KUKA KRL data list: e_fraes_1.dat

&ACCESS RVP2
&REL 8
&COMMENT Fresa C1
&PARAM DISKPATH = KRC:\R1\Program
&PARAM TEMPLATE = C:\KRC\Roboter\Template\vorgabe
&PARAM EDITMASK = *
DEFDAT  e_fraes_1
;FOLD EXTERNAL DECLARATIONS;%{PE}%MKUKATPBASIS,%CEXT,%VCOMMON,%P
;FOLD GRIPPERTECH EXT
EXT  H50 (INT  :IN,INT  :IN,INT  :IN,GRP_TYP  :IN )
;ENDFOLD (GRIPPERTECH EXT)
;FOLD SPOTTECH EXT
EXT  USERSPOT (S_COMMAND  :IN,SPOT_TYPE  :IN )
;ENDFOLD (SPOTTECH EXT)
;FOLD BASISTECH EXT;%{PE}%MKUKATPBASIS,%CEXT,%VEXT,%P
EXT  BAS (BAS_COMMAND  :IN,REAL  :IN )
DECL INT SUCCESS
;ENDFOLD (BASISTECH EXT)
;FOLD USER EXT;%{E}%MKUKATPUSER,%CEXT,%VEXT,%P
;Make your modifications here

;ENDFOLD (USER EXT)
;ENDFOLD (EXTERNAL DECLARATIONS)

DECL E6POS XLHP010={X 388.052307,Y 1486.41003,Z 838.34668,A 150.907806,B -0.182968304,C -18.4479904,S 2,T 3,E1 0.0,E2 0.0,E3 0.0,E4 0.0,E5 0.0,E6 0.0}
DECL FDAT FLHP010={TOOL_NO 1,BASE_NO 0,IPO_FRAME #BASE}
DECL PDAT PPDAT1={VEL 100.0,ACC 100.0,APO_DIST 20.0,APO_MODE #CDIS}
DECL E6POS XLHP015={X 384.866791,Y 1472.83899,Z 444.33551,A -149.197906,B 0.240399107,C -3.14899206,S 18,T 11,E1 0.0,E2 0.0,E3 0.0,E4 0.0,E5 0.0,E6 0.0}
DECL FDAT FLHP015={TOOL_NO 1,BASE_NO 0,IPO_FRAME #BASE}
DECL PDAT PPDAT2={VEL 100.0,ACC 100.0,APO_DIST 10.0}
DECL E6POS XLHP020={X 309.223694,Y 1602.80103,Z 250.550003,A -134.665497,B -0.498555809,C -1.271559,S 18,T 11,E1 0.0,E2 0.0,E3 0.0,E4 0.0,E5 0.0,E6 0.0}
DECL FDAT FLHP020={TOOL_NO 1,BASE_NO 0,IPO_FRAME #BASE}
DECL PDAT PPDAT3={VEL 100.0,ACC 100.0,APO_DIST 5.0,APO_MODE #CDIS}
DECL E6POS XLHP025={X 98.0119705,Y 1699.85095,Z 256.256805,A -134.662704,B -0.490130603,C -1.27114701,S 18,T 11,E1 0.0,E2 0.0,E3 0.0,E4 0.0,E5 0.0,E6 0.0}
DECL FDAT FLHP025={TOOL_NO 1,BASE_NO 0,IPO_FRAME #BASE}
DECL LDAT LCPDAT1={VEL 2.0,ACC 100.0,APO_DIST 2.0,APO_FAC 50.0}
DECL FDAT FDress1={TOOL_NO 1,BASE_NO 0,IPO_FRAME #BASE}
DECL E6POS XDress1={X 99.6608887,Y 1696.71301,Z 300.036499,A -134.662994,B -0.49089241,C -1.27011204,S 18,T 11,E1 0.0,E2 0.0,E3 0.0,E4 0.0,E5 0.0,E6 0.0}
DECL E6POS XPFRESA={X 102.833801,Y 1696.37195,Z 300.660889,A -134.662903,B -0.489995897,C -1.26936698,S 18,T 11,E1 0.0,E2 0.0,E3 0.0,E4 0.0,E5 0.0,E6 0.0}
DECL FDAT Fpfresa={TOOL_NO 1,BASE_NO 0,IPO_FRAME #BASE}
DECL LDAT LCPDAT2={VEL 2.0,ACC 100.0,APO_DIST 100.0,APO_FAC 50.0}
DECL E6POS XLHP030={X 98.0103073,Y 1699.84998,Z 256.256012,A -134.662704,B -0.490198791,C -1.27115798,S 18,T 11,E1 0.0,E2 0.0,E3 0.0,E4 0.0,E5 0.0,E6 0.0}
DECL FDAT FLHP030={TOOL_NO 1,BASE_NO 0,IPO_FRAME #BASE}
DECL LDAT LCPDAT3={VEL 2.0,ACC 100.0,APO_DIST 2.0,APO_FAC 50.0}
DECL E6POS XLHP035={X 154.117096,Y 1756.56104,Z 255.433594,A -134.6642,B -0.492217898,C -1.27078104,S 18,T 11,E1 0.0,E2 0.0,E3 0.0,E4 0.0,E5 0.0,E6 0.0}
DECL FDAT FLHP035={TOOL_NO 1,BASE_NO 0,IPO_FRAME #BASE}
DECL LDAT LCPDAT4={VEL 2.0,ACC 100.0,APO_DIST 10.0,APO_FAC 50.0}
DECL E6POS XLHP040={X 388.047913,Y 1486.42798,Z 838.35553,A 150.914307,B -0.181115806,C -18.4495907,S 18,T 3,E1 0.0,E2 0.0,E3 0.0,E4 0.0,E5 0.0,E6 0.0}
DECL FDAT FLHP040={TOOL_NO 1,BASE_NO 0,IPO_FRAME #BASE}
DECL PDAT PPDAT4={VEL 100.0,ACC 100.0,APO_DIST 15.0}
DECL E6POS XLHP045={X 388.052307,Y 1486.41003,Z 838.34668,A 150.907806,B -0.182964295,C -18.4479904,S 2,T 3,E1 0.0,E2 0.0,E3 0.0,E4 0.0,E5 0.0,E6 0.0}
DECL FDAT FLHP045={TOOL_NO 1,BASE_NO 0,IPO_FRAME #BASE}
DECL PDAT PPDAT5={VEL 100.0,ACC 100.0,APO_DIST 30.0}
DECL SPOT_SUGG_T LAST_SPOT={GUN[] "1                       ",RETR_CMD[] "#OPN                    ",CHOISE[] "#FIRST                  ",CLO_TM[] "1                       ",PGNO1[] "1                       ",PRESS1[] "0                       ",PGNO2[] "1                       ",PRESS2[] "0                       ",SPOT_PARAMS[] "NORMAL                  "}
DECL E6POS XPSOLDA={X 1225.07996,Y 529.649719,Z 849.19989,A 96.8904495,B -6.64519405,C -11.5978298,S 18,T 10,E1 0.0,E2 0.0,E3 0.0,E4 0.0,E5 0.0,E6 0.0}
DECL FDAT FpSOLDA={TOOL_NO 1,BASE_NO 0,IPO_FRAME #BASE}
DECL PDAT PPDAT7={VEL 50.0,ACC 100.0,APO_DIST 100.0}
DECL E6POS XLHP050={X 1225.08105,Y 529.648682,Z 849.200684,A 96.8904419,B -6.64516401,C -11.5979204,S 18,T 10,E1 0.0,E2 0.0,E3 0.0,E4 0.0,E5 0.0,E6 0.0}
DECL FDAT FLHP050={TOOL_NO 1,BASE_NO 0,IPO_FRAME #BASE}
DECL PDAT PPDAT8={VEL 100.0,ACC 80.0,APO_DIST 10.0}
DECL PDAT PPDAT9={VEL 100.0,ACC 100.0,APO_DIST 10.0}
DECL E6POS XLHP005={X 1225.07996,Y 529.636597,Z 849.195007,A 96.8903809,B -6.6447649,C -11.5977697,S 18,T 10,E1 0.0,E2 0.0,E3 0.0,E4 0.0,E5 0.0,E6 0.0}
DECL FDAT FLHP005={TOOL_NO 1,BASE_NO 0,IPO_FRAME #BASE,TQ_STATE FALSE}
DECL FDAT FDress2={TOOL_NO 1,BASE_NO 0,IPO_FRAME #BASE}
DECL E6POS XDress2={X 251.336395,Y 1645.68506,Z 283.317688,A 178.927307,B -0.849079311,C -0.868841827,S 18,T 11,E1 0.0,E2 0.0,E3 0.0,E4 0.0,E5 0.0,E6 0.0}
DECL BASIS_SUGG_T LAST_BASIS={POINT1[] "P5                      ",POINT2[] "P5                      ",CP_PARAMS[] "CPDAT7                  ",PTP_PARAMS[] "PDAT10                  ",CONT[] "C_DIS                   ",CP_VEL[] "0.5                     ",PTP_VEL[] "80                      ",SYNC_PARAMS[] "SYNCDAT                 ",SPL_NAME[] "S0                      "}
DECL E6POS XP1={X 382.214813,Y 1646.07104,Z 258.947113,A 178.9245,B -0.858626127,C -0.883606017,S 18,T 11,E1 0.0,E2 0.0,E3 0.0,E4 0.0,E5 0.0,E6 0.0}
DECL FDAT FP1={TOOL_NO 1,BASE_NO 0,IPO_FRAME #BASE,POINT2[] " ",TQ_STATE FALSE}
DECL LDAT LCPDAT5={VEL 2.0,ACC 100.0,APO_DIST 100.0,APO_FAC 50.0,AXIS_VEL 100.0,AXIS_ACC 100.0,ORI_TYP #VAR,CIRC_TYP #BASE,JERK_FAC 50.0,GEAR_JERK 50.0,EXAX_IGN 0}
DECL E6POS XP2={X 255.032104,Y 1646.46802,Z 239.541595,A 178.911499,B -0.883683383,C -0.972572982,S 18,T 11,E1 0.0,E2 0.0,E3 0.0,E4 0.0,E5 0.0,E6 0.0}
DECL FDAT FP2={TOOL_NO 1,BASE_NO 0,IPO_FRAME #BASE,POINT2[] " ",TQ_STATE FALSE}
DECL LDAT LCPDAT6={VEL 2.0,ACC 100.0,APO_DIST 100.0,APO_FAC 50.0,AXIS_VEL 100.0,AXIS_ACC 100.0,ORI_TYP #VAR,CIRC_TYP #BASE,JERK_FAC 50.0,GEAR_JERK 50.0,EXAX_IGN 0}
DECL E6POS XP3={X 154.117096,Y 1756.56104,Z 255.433594,A -134.664093,B -0.492220193,C -1.27076995,S 18,T 11,E1 0.0,E2 0.0,E3 0.0,E4 0.0,E5 0.0,E6 0.0}
DECL FDAT FP3={TOOL_NO 1,BASE_NO 0,IPO_FRAME #BASE,POINT2[] " ",TQ_STATE FALSE}
DECL LDAT LCPDAT7={VEL 2.0,ACC 100.0,APO_DIST 100.0,APO_FAC 50.0,AXIS_VEL 100.0,AXIS_ACC 100.0,ORI_TYP #VAR,CIRC_TYP #BASE,JERK_FAC 50.0,GEAR_JERK 50.0,EXAX_IGN 0}
DECL E6POS XP4={X 384.877106,Y 1472.83899,Z 444.332214,A -149.197906,B 0.240724206,C -3.14874506,S 18,T 11,E1 0.0,E2 0.0,E3 0.0,E4 0.0,E5 0.0,E6 0.0}
DECL FDAT FP4={TOOL_NO 1,BASE_NO 0,IPO_FRAME #BASE,POINT2[] " ",TQ_STATE FALSE}
DECL PDAT PPDAT6={VEL 100.0,ACC 100.0,APO_DIST 10.0,APO_MODE #CDIS,GEAR_JERK 50.0}
DECL E6POS XP5={X 309.234985,Y 1602.80005,Z 250.546005,A -134.665298,B -0.498314798,C -1.27121103,S 18,T 11,E1 0.0,E2 0.0,E3 0.0,E4 0.0,E5 0.0,E6 0.0}
DECL FDAT FP5={TOOL_NO 1,BASE_NO 0,IPO_FRAME #BASE,POINT2[] " ",TQ_STATE FALSE}
DECL PDAT PPDAT10={VEL 100.0,ACC 100.0,APO_DIST 10.0,APO_MODE #CDIS,GEAR_JERK 50.0}
DECL PDAT PPDAT11={VEL 50.0,ACC 100.0,APO_DIST 100.0}
ENDDAT
